TYPE ST_TwinSAFE :
STRUCT
	
///////////////////////////////////////////////////////////////////////////Safety OUTPUTS///////////////////////////////////////////////////////////////////////////////////////
	
	iErrorAcknowledge               		AT %Q*			: 	BOOL;	
	iProcessDoorClosing              		AT %Q*			: 	BOOL;	
	iAirPressureMaxValue					AT %Q*			: 	UINT;
	iAirPressureMinValue					AT %Q*			: 	UINT;
	iAirSupplyMeasurement					AT %Q*			: 	UINT;
	iProcessDoorClosedCondition				AT %Q*			: 	BOOL;	
	
///////////////////////////////////////////////////////////////////////////Safety Inputs///////////////////////////////////////////////////////////////////////////////////////	

	qAirErrorSignal							AT %I*			: 	BOOL;	
	qAirPressureAbove						AT %I*			: 	BOOL;	
	qAirPressureBelow						AT %I*			: 	BOOL;	
	qProcessDoorClosed						AT %I*			: 	BOOL;	
	qSafetyOk								AT %I*			: 	BOOL;	
	qStartProcessSignal						AT %I*			: 	BOOL;
	qE_StopPressed							AT %I*			: 	BOOL;	
	qMainDoorOpened							AT %I*			: 	BOOL;
	qProcessDoorSafe						AT %I*			: 	BOOL;
	qTwoHandsSafe							AT %I*			: 	BOOL;

END_STRUCT
END_TYPE

(* stored: Version 1.1.0.1, ProductVersion 3.1.4024.13
   DUT ST_TwinSAFE: Id {53872549-54d4-4379-ac97-82f6a4774545} *)
